FUNCTION_BLOCK Adaptive_Threshold (* openCV adaptive threshold *)
  (* Version 1.0, AN, SWDC RTSoft *)
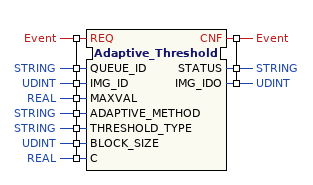
  EVENT_INPUT
    REQ WITH QUEUE_ID, IMG_ID, MAXVAL, ADAPTIVE_METHOD, THRESHOLD_TYPE, BLOCK_SIZE, C;
  END_EVENT
  EVENT_OUTPUT
    CNF WITH STATUS, IMG_IDO;
  END_EVENT
  VAR_INPUT
    QUEUE_ID : STRING;
    IMG_ID : UDINT;
    MAXVAL : REAL;
    ADAPTIVE_METHOD : STRING;
    THRESHOLD_TYPE : STRING;
    BLOCK_SIZE : UDINT;
    C : REAL;
  END_VAR
  VAR_OUTPUT
    STATUS : STRING;
    IMG_IDO : UDINT;
  END_VAR
  ALGORITHM REQ IN ST:

  END_ALGORITHM
END_FUNCTION_BLOCK
